(* IEC 61131-3 sources: A_BST22/, 17 files *)

(* ---- PLC_Arcade_System_ST.st ---- *)
// Sysmac Studio Structured Text - PLC Arcade System
// Omron NX102 PLC Implementation

// Global Variables Declaration
VAR_GLOBAL
    // ============================================================================
    // INPUT MAPPING (Contacts)
    // ============================================================================
    IBTN_R AT %IX0.0: BOOL;      // Red button - DI0
    IBTN_B AT %IX0.2: BOOL;      // Blue button - DI2
    IBTN_Y AT %IX0.4: BOOL;      // Yellow button - DI4
    ISEL_LT AT %IX0.3: BOOL;     // Simon Says selector - DI3 (Yellow wire)
    ISEL_R AT %IX0.5: BOOL;      // Reaction Game selector - DI5 (Green wire)
    IBTN_M AT %IX0.1: BOOL;      // Main button - DI1 (Brown wire)

    // ============================================================================
    // OUTPUT MAPPING (LEDs)
    // ============================================================================
    OLED_R AT %QX0.1: BOOL;      // Red LED - DO1
    OLED_B AT %QX0.3: BOOL;      // Blue LED - DO3
    OLED_Y AT %QX0.5: BOOL;      // Yellow LED - DO5
    OLED_MAIN AT %QX0.0: BOOL;   // Main LED - DO0 (White wire)

    // ============================================================================
    // SYSTEM CONTROL VARIABLES
    // ============================================================================
    SystemActive: BOOL := FALSE;
    GameRunning: BOOL := FALSE;
    ModeLocked: BOOL := FALSE;
    EmergencyStop: BOOL := FALSE;

    // Mode Selection
    CurrentMode: INT := 0;  // 0=Simon Says, 1=Reaction Game, 2=Idle
    PreviousMode: INT := 0;

    // Button States (Debounced)
    BtnR_State: BOOL := FALSE;
    BtnB_State: BOOL := FALSE;
    BtnY_State: BOOL := FALSE;
    BtnM_State: BOOL := FALSE;

    // Button Edge Detection
    BtnR_Rising: BOOL := FALSE;
    BtnB_Rising: BOOL := FALSE;
    BtnY_Rising: BOOL := FALSE;
    BtnM_Rising: BOOL := FALSE;

    // Previous Button States for Edge Detection
    PrevBtnR: BOOL := FALSE;
    PrevBtnB: BOOL := FALSE;
    PrevBtnY: BOOL := FALSE;
    PrevBtnM: BOOL := FALSE;

    // ============================================================================
    // DEBOUNCE TIMERS (Sysmac Studio TON)
    // ============================================================================
    DebounceTimer: TON;
    ModeLockTimer: TON;

    // ============================================================================
    // CONTINUOUS RANDOM GENERATOR VARIABLES
    // ============================================================================
    RandomGenActive: BOOL := FALSE;
    RandomGenRunning: BOOL := FALSE;
    RandomCounter: INT := 0;
    OutputSelect: INT := 0;

    // Random Generator Outputs
    RandomOut1: BOOL := FALSE;
    RandomOut2: BOOL := FALSE;
    RandomOut3: BOOL := FALSE;

    // ============================================================================
    // SIMON SAYS GAME VARIABLES
    // ============================================================================
    SimonActive: BOOL := FALSE;
    SimonGameOver: BOOL := FALSE;
    SimonState: INT := 0;  // 0=Off, 1=Init, 2=Generate, 3=Show, 4=Input, 5=Check, 6=Complete

    SimonSequence: ARRAY[1..20] OF INT := [0,0,0,0,0,0,0,0,0,0,0,0,0,0,0,0,0,0,0,0];
    SequenceLength: INT := 1;
    CurrentStep: INT := 0;
    PlayerInputStep: INT := 0;

    SimonScore: INT := 0;
    SimonLevel: INT := 1;

    // Simon Says Timers
    SimonSequenceTimer: TON;
    SimonInputTimer: TON;
    SimonPauseTimer: TON;

    // Simon Says Outputs
    SimonOut1: BOOL := FALSE;
    SimonOut2: BOOL := FALSE;
    SimonOut3: BOOL := FALSE;

    // ============================================================================
    // REACTION GAME VARIABLES
    // ============================================================================
    ReactionActive: BOOL := FALSE;
    ReactionGameOver: BOOL := FALSE;
    ReactionState: INT := 0;  // 0=Off, 1=Wait, 2=Show, 3=Score

    ReactionStartTime: INT := 0;
    ReactionEndTime: INT := 0;
    ReactionScore: INT := 0;
    ReactionTarget: INT := 0;  // Which LED to light up (1,2,3)

    // Reaction Game Timers
    ReactionWaitTimer: TON;
    ReactionShowTimer: TON;

    // Reaction Game Outputs
    ReactionOut1: BOOL := FALSE;
    ReactionOut2: BOOL := FALSE;
    ReactionOut3: BOOL := FALSE;

    // ============================================================================
    // OUTPUT MAPPER VARIABLES
    // ============================================================================
    OutputPriority: INT := 0;  // 0=Off, 1=Game, 2=Status, 3=Emergency
    OutputConflict: BOOL := FALSE;
    SafetyInterlock: BOOL := TRUE;
    SystemHealthy: BOOL := TRUE;

    // Status Outputs
    StatusOut1: BOOL := FALSE;
    StatusOut2: BOOL := FALSE;
    StatusOut3: BOOL := FALSE;

    // Emergency Outputs
    EmergencyOut1: BOOL := FALSE;
    EmergencyOut2: BOOL := FALSE;
    EmergencyOut3: BOOL := FALSE;

    // ============================================================================
    // TIMING VARIABLES (Sysmac Studio TON)
    // ============================================================================
    SystemTimer: TON;
    BlinkTimer: TON;

    // ============================================================================
    // DIAGNOSTIC VARIABLES
    // ============================================================================
    ConflictCounter: INT := 0;
    SafetyFailureCounter: INT := 0;
    SystemFailureCounter: INT := 0;

END_VAR

// ============================================================================
// MAIN PROGRAM LOGIC
// ============================================================================

// Note: Input mapping is done directly in VAR_GLOBAL with AT %IX addresses
// No additional mapping needed - inputs are automatically read from hardware

// Button Edge Detection
BtnR_Rising := IBTN_R AND NOT PrevBtnR;
BtnB_Rising := IBTN_B AND NOT PrevBtnB;
BtnY_Rising := IBTN_Y AND NOT PrevBtnY;
BtnM_Rising := IBTN_M AND NOT PrevBtnM;

PrevBtnR := IBTN_R;
PrevBtnB := IBTN_B;
PrevBtnY := IBTN_Y;
PrevBtnM := IBTN_M;

// Button Debouncing (Sysmac Studio TON syntax)
DebounceTimer(IN := IBTN_R OR IBTN_B OR IBTN_Y OR IBTN_M, PT := T#50MS);

IF DebounceTimer.Q THEN
    BtnR_State := IBTN_R;
    BtnB_State := IBTN_B;
    BtnY_State := IBTN_Y;
    BtnM_State := IBTN_M;
    DebounceTimer(IN := FALSE, PT := T#0MS);  // Reset timer
END_IF;

// Mode Selection Logic
PreviousMode := CurrentMode;

IF ISEL_LT THEN
    CurrentMode := 0;  // Simon Says
ELSIF ISEL_R THEN
    CurrentMode := 1;  // Reaction Game
ELSE
    CurrentMode := 2;  // Idle Mode
END_IF;

// Mode Lock Logic
IF BtnM_Rising AND NOT ModeLocked THEN
    ModeLocked := TRUE;
    ModeLockTimer(IN := FALSE, PT := T#0MS);
ELSIF BtnM_Rising AND ModeLocked THEN
    ModeLocked := FALSE;
END_IF;

// System Activation
IF ModeLocked AND BtnM_Rising THEN
    GameRunning := TRUE;
    SystemActive := TRUE;
END_IF;

// Emergency Stop
IF EmergencyStop THEN
    GameRunning := FALSE;
    SystemActive := FALSE;
    ModeLocked := FALSE;
    OutputPriority := 3;  // Emergency priority
END_IF;

// ============================================================================
// CONTINUOUS RANDOM GENERATOR
// ============================================================================

RandomGenActive := SystemActive;

// Random Generator Timer (Sysmac Studio TON syntax)
SystemTimer(IN := RandomGenActive, PT := T#100MS);

// Increment Counter
IF SystemTimer.Q THEN
    SystemTimer(IN := FALSE, PT := T#0MS);  // Reset timer
    RandomCounter := RandomCounter + 1;
    IF RandomCounter >= 1000 THEN
        RandomCounter := 0;
    END_IF;
END_IF;

// Calculate Output Selection
OutputSelect := RandomCounter MOD 3;
RandomGenRunning := RandomGenActive;

// Set Random Outputs
RandomOut1 := RandomGenRunning AND (OutputSelect = 0);
RandomOut2 := RandomGenRunning AND (OutputSelect = 1);
RandomOut3 := RandomGenRunning AND (OutputSelect = 2);

// ============================================================================
// SIMON SAYS GAME LOGIC
// ============================================================================

SimonActive := (CurrentMode = 0) AND GameRunning;

// Simon Says State Machine
CASE SimonState OF
    0:  // Game Off
        IF SimonActive THEN
            SimonState := 1;
            SimonScore := 0;
            SimonLevel := 1;
            SequenceLength := 1;
            SimonGameOver := FALSE;
        END_IF;

    1:  // Initialize Game
        CurrentStep := 0;
        PlayerInputStep := 0;
        SimonSequenceTimer(IN := FALSE, PT := T#0MS);
        SimonInputTimer(IN := FALSE, PT := T#0MS);
        SimonPauseTimer(IN := FALSE, PT := T#0MS);
        SimonState := 2;

    2:  // Generate Sequence
        FOR i := 1 TO SequenceLength DO
            SimonSequence[i] := (RandomCounter + i) MOD 3 + 1;
        END_FOR;
        SimonState := 3;

    3:  // Show Sequence
        IF CurrentStep < SequenceLength THEN
            SimonSequenceTimer(IN := TRUE, PT := T#500MS);
            IF SimonSequenceTimer.Q THEN
                SimonSequenceTimer(IN := FALSE, PT := T#0MS);  // Reset timer
                CurrentStep := CurrentStep + 1;
            END_IF;
        ELSE
            SimonPauseTimer(IN := TRUE, PT := T#1000MS);
            IF SimonPauseTimer.Q THEN
                SimonPauseTimer(IN := FALSE, PT := T#0MS);  // Reset timer
                CurrentStep := 0;
                PlayerInputStep := 0;
                SimonState := 4;
            END_IF;
        END_IF;

    4:  // Wait for Player Input
        SimonInputTimer(IN := TRUE, PT := T#5000MS);

        // Check for player input
        IF BtnR_Rising THEN
            IF SimonSequence[PlayerInputStep + 1] = 1 THEN
                PlayerInputStep := PlayerInputStep + 1;
            ELSE
                SimonGameOver := TRUE;
                SimonState := 6;
            END_IF;
        ELSIF BtnB_Rising THEN
            IF SimonSequence[PlayerInputStep + 1] = 2 THEN
                PlayerInputStep := PlayerInputStep + 1;
            ELSE
                SimonGameOver := TRUE;
                SimonState := 6;
            END_IF;
        ELSIF BtnY_Rising THEN
            IF SimonSequence[PlayerInputStep + 1] = 3 THEN
                PlayerInputStep := PlayerInputStep + 1;
            ELSE
                SimonGameOver := TRUE;
                SimonState := 6;
            END_IF;
        END_IF;

        // Check if input complete or timeout
        IF PlayerInputStep >= SequenceLength THEN
            SimonScore := SimonScore + (SequenceLength * 10);
            SequenceLength := SequenceLength + 1;
            SimonState := 2;  // Generate next sequence
        ELSIF SimonInputTimer.Q THEN
            SimonGameOver := TRUE;
            SimonState := 6;
        END_IF;

    5:  // Check Input (Not used in this implementation)
        SimonState := 6;

    6:  // Game Complete
        SimonInputTimer(IN := FALSE, PT := T#0MS);  // Reset timer
        IF NOT SimonActive THEN
            SimonState := 0;
        END_IF;
END_CASE;

// Simon Says Output Control
SimonOut1 := (SimonState = 3) AND (CurrentStep <= SequenceLength) AND (SimonSequence[CurrentStep] = 1);
SimonOut2 := (SimonState = 3) AND (CurrentStep <= SequenceLength) AND (SimonSequence[CurrentStep] = 2);
SimonOut3 := (SimonState = 3) AND (CurrentStep <= SequenceLength) AND (SimonSequence[CurrentStep] = 3);

// Add player input feedback
SimonOut1 := SimonOut1 OR ((SimonState = 4) AND BtnR_State);
SimonOut2 := SimonOut2 OR ((SimonState = 4) AND BtnB_State);
SimonOut3 := SimonOut3 OR ((SimonState = 4) AND BtnY_State);

// ============================================================================
// REACTION GAME LOGIC
// ============================================================================

ReactionActive := (CurrentMode = 1) AND GameRunning;

// Reaction Game State Machine
CASE ReactionState OF
    0:  // Game Off
        IF ReactionActive THEN
            ReactionState := 1;
            ReactionScore := 0;
            ReactionGameOver := FALSE;
        END_IF;

    1:  // Wait Phase
        ReactionWaitTimer(IN := TRUE, PT := T#2000MS + (RandomCounter MOD 3000MS));
        IF ReactionWaitTimer.Q THEN
            ReactionWaitTimer(IN := FALSE, PT := T#0MS);  // Reset timer
            ReactionTarget := (RandomCounter MOD 3) + 1;
            ReactionState := 2;
        END_IF;

    2:  // Show Target
        ReactionShowTimer(IN := TRUE, PT := T#1000MS);

        // Check for player reaction
        IF (ReactionTarget = 1) AND BtnR_Rising THEN
            ReactionEndTime := 1000 - ReactionShowTimer.ET;
            ReactionScore := ReactionEndTime;
            ReactionState := 3;
        ELSIF (ReactionTarget = 2) AND BtnB_Rising THEN
            ReactionEndTime := 1000 - ReactionShowTimer.ET;
            ReactionScore := ReactionEndTime;
            ReactionState := 3;
        ELSIF (ReactionTarget = 3) AND BtnY_Rising THEN
            ReactionEndTime := 1000 - ReactionShowTimer.ET;
            ReactionScore := ReactionEndTime;
            ReactionState := 3;
        ELSIF ReactionShowTimer.Q THEN
            ReactionGameOver := TRUE;
            ReactionState := 3;
        END_IF;

    3:  // Score Phase
        IF NOT ReactionActive THEN
            ReactionState := 0;
        ELSIF BtnM_Rising THEN
            ReactionState := 1;  // Start new round
        END_IF;
END_CASE;

// Reaction Game Output Control
ReactionOut1 := (ReactionState = 2) AND (ReactionTarget = 1);
ReactionOut2 := (ReactionState = 2) AND (ReactionTarget = 2);
ReactionOut3 := (ReactionState = 2) AND (ReactionTarget = 3);

// ============================================================================
// OUTPUT MAPPER AND SAFETY LOGIC
// ============================================================================

// Detect Output Conflicts
OutputConflict := (SimonActive AND ReactionActive) OR
                  (SimonActive AND (CurrentMode = 2)) OR
                  (ReactionActive AND (CurrentMode = 2));

// Output Priority Control
IF EmergencyStop THEN
    OutputPriority := 3;  // Emergency
ELSIF NOT SystemHealthy THEN
    OutputPriority := 3;  // Emergency
ELSIF OutputConflict THEN
    OutputPriority := 3;  // Emergency
ELSIF GameRunning THEN
    OutputPriority := 1;  // Game
ELSIF SystemActive THEN
    OutputPriority := 2;  // Status
ELSE
    OutputPriority := 0;  // Off
END_IF;

// Status Outputs
StatusOut1 := SystemActive;
StatusOut2 := GameRunning;
StatusOut3 := OutputConflict OR NOT SystemHealthy;

// Emergency Outputs
EmergencyOut1 := EmergencyStop;
EmergencyOut2 := NOT SystemHealthy;
EmergencyOut3 := OutputConflict;

// Final Output Mapping
CASE OutputPriority OF
    0:  // System Off
        OLED_R := FALSE;
        OLED_B := FALSE;
        OLED_Y := FALSE;
        OLED_MAIN := FALSE;

    1:  // Game Outputs
        IF CurrentMode = 0 THEN  // Simon Says
            OLED_R := SimonOut1;
            OLED_B := SimonOut2;
            OLED_Y := SimonOut3;
        ELSIF CurrentMode = 1 THEN  // Reaction Game
            OLED_R := ReactionOut1;
            OLED_B := ReactionOut2;
            OLED_Y := ReactionOut3;
        ELSE  // Idle Mode
            OLED_R := RandomOut1;
            OLED_B := RandomOut2;
            OLED_Y := RandomOut3;
        END_IF;
        OLED_MAIN := GameRunning;

    2:  // Status Outputs
        OLED_R := StatusOut1;
        OLED_B := StatusOut2;
        OLED_Y := StatusOut3;
        OLED_MAIN := ModeLocked;

    3:  // Emergency Outputs
        OLED_R := EmergencyOut1;
        OLED_B := EmergencyOut2;
        OLED_Y := EmergencyOut3;
        OLED_MAIN := FALSE;
END_CASE;

// Note: Output mapping is done directly in VAR_GLOBAL with AT %QX addresses
// No additional mapping needed - outputs are automatically written to hardware
// OLED_R AT %QX0.1, OLED_B AT %QX0.3, OLED_Y AT %QX0.5, OLED_MAIN AT %QX0.0

// ============================================================================
// DIAGNOSTIC AND MONITORING
// ============================================================================

// Count Conflicts
IF OutputConflict THEN
    ConflictCounter := ConflictCounter + 1;
END_IF;

// Count Safety Failures
IF NOT SystemHealthy THEN
    SafetyFailureCounter := SafetyFailureCounter + 1;
END_IF;

// System Health Check
SystemHealthy := TRUE;  // Placeholder - implement actual health checks

// ============================================================================
// END OF PROGRAM
// ============================================================================

(* ---- HandleButtonPress.st ---- *)
FUNCTION HandleButtonPress : BOOL
VAR_INPUT
    ButtonPressed : BOOL;           // TRUE if this button was pressed
    ExpectedLED : INT;             // The LED number that should be lit (1=Yellow, 2=Blue, 3=Red)
    CurrentLED : INT;              // The currently lit LED number
END_VAR

VAR_IN_OUT
    Score : INT;                   // Player's current score
    GameActive : BOOL;             // Game state flag
    GameOver_Active : BOOL;        // Game over state flag
    LEDActive : BOOL;              // LED phase active flag
    GapActive : BOOL;              // Gap phase active flag
    HighScore : INT;               // High score tracking
    GameOver_Step : INT;           // Game over sequence step
    T_LED_On : TON;                // LED timer
    T_Gap : TON;                   // Gap timer
    T_Seq : TON;                   // Sequence timer
    Rand_Gen : FB_Random;          // Random number generator
    RandN : REAL;                  // Random number output
END_VAR

// Function returns TRUE if button was handled (pressed)
HandleButtonPress := ButtonPressed;

IF ButtonPressed THEN
    IF CurrentLED = ExpectedLED THEN
        // Correct button pressed - add point and continue
        Score := Score + 1;
        LEDActive := FALSE;
        GapActive := TRUE;
        T_LED_On(IN := FALSE);

        // Generate next random gap duration
        Rand_Gen(Execute := TRUE, Seed := 0, Rnd => RandN);
        T_Gap(IN := FALSE);
        IF RandN < 0.2 THEN
            T_Gap(PT := t#500ms);
        ELSIF RandN < 0.4 THEN
            T_Gap(PT := t#750ms);
        ELSIF RandN < 0.6 THEN
            T_Gap(PT := t#1000ms);
        ELSIF RandN < 0.8 THEN
            T_Gap(PT := t#1250ms);
        ELSE
            T_Gap(PT := t#1500ms);
        END_IF;
    ELSE
        // Wrong button pressed - game over
        GameActive := FALSE;
        GameOver_Active := TRUE;
        GameOver_Step := 0;
        T_Seq(IN := FALSE, PT := t#300ms);
        LEDActive := FALSE;
        GapActive := FALSE;
        T_LED_On(IN := FALSE);
        T_Gap(IN := FALSE);

        // Update high score if needed
        IF Score > HighScore THEN
            HighScore := Score;
        END_IF;
    END_IF;
END_IF;

END_FUNCTION

(* ---- FB_CheckButtonPress.st ---- *)
FUNCTION_BLOCK FB_CheckButtonPress
VAR_INPUT
    ButtonPressed : BOOL;          // Trigger for this button
    ExpectedLED : INT;             // Which LED should be lit (1=Yellow, 2=Blue, 3=Red)
    CurrentLED : INT;              // Which LED is actually lit
    Score : INT;                   // Current score
    HighScore : INT;               // Current high score
END_VAR

VAR_OUTPUT
    IsCorrect : BOOL;              // TRUE if correct button pressed
    IsWrong : BOOL;                // TRUE if wrong button pressed
    NewScore : INT;                // Updated score
    NewHighScore : INT;            // Updated high score
    NextGapTime : TIME;            // Random gap time for next round
    EndGame : BOOL;                // Signal to end the game
    ContinueGame : BOOL;           // Signal to continue to next round
END_VAR

VAR
    Rand_Gen : FB_RandomGenerator; // Random number generator (adjust to your actual FB name)
    RandN : REAL;
END_VAR

// Initialize outputs
IsCorrect := FALSE;
IsWrong := FALSE;
NewScore := Score;
NewHighScore := HighScore;
EndGame := FALSE;
ContinueGame := FALSE;

// Check if button was pressed
IF ButtonPressed THEN
    // Check if it's the correct button
    IF CurrentLED = ExpectedLED THEN
        // Correct button pressed
        IsCorrect := TRUE;
        ContinueGame := TRUE;
        NewScore := Score + 1;

        // Generate next random gap time
        Rand_Gen(Execute := TRUE, Seed := 0, Rnd => RandN);
        IF RandN < 0.2 THEN
            NextGapTime := t#500ms;
        ELSIF RandN < 0.4 THEN
            NextGapTime := t#750ms;
        ELSIF RandN < 0.6 THEN
            NextGapTime := t#1000ms;
        ELSIF RandN < 0.8 THEN
            NextGapTime := t#1250ms;
        ELSE
            NextGapTime := t#1500ms;
        END_IF;
    ELSE
        // Wrong button pressed - game over
        IsWrong := TRUE;
        EndGame := TRUE;

        // Update high score if needed
        IF Score > HighScore THEN
            NewHighScore := Score;
        ELSE
            NewHighScore := HighScore;
        END_IF;
    END_IF;
END_IF;

END_FUNCTION_BLOCK

(* ---- FB_RandomGenerator.st ---- *)
(* ====================================================================
   FUNCTION BLOCK: Random Number Generator for Simon Says
   Generates pseudo-random numbers 1-3 for button selection
   ==================================================================== *)

FUNCTION_BLOCK FB_RandomGenerator
VAR_INPUT
    Generate : BOOL;        (* Trigger to generate new random number *)
    Reset : BOOL;           (* Reset seed to initial value *)
    MaxValue : INT := 3;    (* Maximum value (3 for 3 buttons, 4 for 4 buttons) *)
END_VAR

VAR_OUTPUT
    RandomValue : INT;      (* Output: 1 to MaxValue *)
    Done : BOOL;           (* Pulse when new number generated *)
END_VAR

VAR
    Seed : DINT := 12345;  (* Internal seed value *)
    LastGenerate : BOOL;   (* Edge detection *)
    PulseTimer : TON;      (* Timer for done pulse *)
END_VAR

(* Reset seed if requested *)
IF Reset THEN
    Seed := 12345;
    RandomValue := 0;
    Done := FALSE;
END_IF;

(* Detect rising edge of Generate signal *)
IF Generate AND NOT LastGenerate THEN
    (* Linear Congruential Generator algorithm *)
    Seed := (Seed * 1103515245 + 12345) MOD 2147483648;

    (* Convert to desired range (1 to MaxValue) *)
    RandomValue := (ABS(Seed) MOD MaxValue) + 1;

    (* Trigger done pulse *)
    Done := TRUE;
    PulseTimer(IN := TRUE, PT := T#100MS);
END_IF;

(* Clear done pulse after timer *)
PulseTimer(IN := PulseTimer.IN, PT := T#100MS);
IF PulseTimer.Q THEN
    Done := FALSE;
    PulseTimer(IN := FALSE);
END_IF;

(* Update edge detection *)
LastGenerate := Generate;

END_FUNCTION_BLOCK

(* ---- FB_SimonSays.st ---- *)
(* ====================================================================== *)
(* Function Block: FB_SimonSays                                          *)
(* Simon Says Game Logic for Omron NX102                                *)
(* ====================================================================== *)

FUNCTION_BLOCK FB_SimonSays

VAR_INPUT
    (* Button Inputs *)
    i_YellowButton : BOOL;     (* Yellow button contact *)
    i_BlueButton : BOOL;       (* Blue button contact *)
    i_RedButton : BOOL;         (* Red button contact *)
    i_StartButton : BOOL;       (* Start/Stop button *)
    i_Reset : BOOL;             (* Reset game *)

    (* Game Parameters *)
    i_MaxLevel : INT := 10;    (* Maximum sequence length *)
    i_ShowTime : TIME := T#500MS;   (* LED display time *)
    i_GapTime : TIME := T#200MS;    (* Gap between LEDs *)
    i_InputTimeout : TIME := T#3S;  (* Player input timeout *)
END_VAR

VAR_OUTPUT
    (* LED Outputs *)
    q_YellowLED : BOOL;        (* Yellow button LED *)
    q_BlueLED : BOOL;          (* Blue button LED *)
    q_RedLED : BOOL;           (* Red button LED *)

    (* Status Outputs *)
    q_GameActive : BOOL;        (* Game is active *)
    q_CurrentLevel : INT;       (* Current level *)
    q_GameWon : BOOL;          (* Player won *)
    q_GameLost : BOOL;         (* Player lost *)
    q_State : INT;             (* Current state for diagnostics *)
END_VAR

VAR
    (* Internal State Machine *)
    State : INT := 0;
    NextState : INT := 0;

    (* Sequence Storage *)
    Sequence : ARRAY[0..49] OF INT;
    Level : INT := 0;
    SeqIndex : INT := 0;
    InputIndex : INT := 0;

    (* Timers *)
    tmr_Show : TON;
    tmr_Gap : TON;
    tmr_Input : TON;
    tmr_GameOver : TON;
    tmr_Blink : TON;

    (* Edge Detection *)
    rtrig_Yellow : R_TRIG;
    rtrig_Blue : R_TRIG;
    rtrig_Red : R_TRIG;
    rtrig_Start : R_TRIG;

    (* Flags *)
    ShowingLED : BOOL := FALSE;
    InGap : BOOL := FALSE;
    InputReceived : BOOL := FALSE;
    CorrectInput : BOOL := FALSE;

    (* Random Generation *)
    RandomSeed : DINT := 0;
    RandomValue : INT := 0;

    (* Temporary Variables *)
    i : INT;
    BlinkState : BOOL := FALSE;
END_VAR

(* ====================================================================== *)
(* MAIN LOGIC                                                            *)
(* ====================================================================== *)

(* Edge Detection *)
rtrig_Yellow(CLK := i_YellowButton);
rtrig_Blue(CLK := i_BlueButton);
rtrig_Red(CLK := i_RedButton);
rtrig_Start(CLK := i_StartButton);

(* Update Random Seed *)
RandomSeed := RandomSeed + 1;
IF RandomSeed > 100000 THEN
    RandomSeed := 1;
END_IF;

(* Reset Logic *)
IF i_Reset THEN
    State := 0;
    Level := 0;
    SeqIndex := 0;
    InputIndex := 0;
    q_YellowLED := FALSE;
    q_BlueLED := FALSE;
    q_RedLED := FALSE;
    q_GameActive := FALSE;
    q_GameWon := FALSE;
    q_GameLost := FALSE;
    ShowingLED := FALSE;
    InGap := FALSE;
    RETURN;
END_IF;

(* State Machine *)
CASE State OF

    (* ====================================================================== *)
    0: (* IDLE STATE *)
    (* ====================================================================== *)
        q_GameActive := FALSE;
        q_YellowLED := FALSE;
        q_BlueLED := FALSE;
        q_RedLED := FALSE;
        q_GameWon := FALSE;
        q_GameLost := FALSE;

        IF rtrig_Start.Q THEN
            (* Initialize new game *)
            Level := 1;
            SeqIndex := 0;
            InputIndex := 0;

            (* Generate first random button *)
            RandomValue := INT(RandomSeed MOD 3) + 1;
            Sequence[0] := RandomValue;

            (* Start game *)
            q_GameActive := TRUE;
            State := 1;
        END_IF;

    (* ====================================================================== *)
    1: (* SHOW SEQUENCE STATE *)
    (* ====================================================================== *)
        IF SeqIndex < Level THEN
            IF NOT ShowingLED AND NOT InGap THEN
                (* Start showing next LED *)
                ShowingLED := TRUE;
                tmr_Show(IN := FALSE);
                tmr_Show(IN := TRUE, PT := i_ShowTime);

                (* Turn on appropriate LED *)
                CASE Sequence[SeqIndex] OF
                    1: q_YellowLED := TRUE;
                    2: q_BlueLED := TRUE;
                    3: q_RedLED := TRUE;
                END_CASE;
            END_IF;

            (* Handle LED display timing *)
            IF ShowingLED THEN
                tmr_Show(IN := TRUE, PT := i_ShowTime);
                IF tmr_Show.Q THEN
                    (* Turn off LEDs *)
                    q_YellowLED := FALSE;
                    q_BlueLED := FALSE;
                    q_RedLED := FALSE;
                    ShowingLED := FALSE;
                    InGap := TRUE;
                    tmr_Gap(IN := FALSE);
                    tmr_Gap(IN := TRUE, PT := i_GapTime);
                END_IF;
            END_IF;

            (* Handle gap timing *)
            IF InGap THEN
                tmr_Gap(IN := TRUE, PT := i_GapTime);
                IF tmr_Gap.Q THEN
                    InGap := FALSE;
                    SeqIndex := SeqIndex + 1;
                END_IF;
            END_IF;
        ELSE
            (* Sequence display complete *)
            SeqIndex := 0;
            InputIndex := 0;
            State := 2;
            tmr_Input(IN := FALSE);
            tmr_Input(IN := TRUE, PT := i_InputTimeout);
        END_IF;

    (* ====================================================================== *)
    2: (* WAIT FOR PLAYER INPUT STATE *)
    (* ====================================================================== *)
        (* Check for timeout *)
        tmr_Input(IN := TRUE, PT := i_InputTimeout);
        IF tmr_Input.Q THEN
            (* Timeout - player loses *)
            State := 4;
            tmr_GameOver(IN := FALSE);
            tmr_GameOver(IN := TRUE, PT := T#2S);
        END_IF;

        (* Process button inputs *)
        InputReceived := FALSE;
        CorrectInput := FALSE;

        IF rtrig_Yellow.Q THEN
            InputReceived := TRUE;
            q_YellowLED := TRUE;
            IF Sequence[InputIndex] = 1 THEN
                CorrectInput := TRUE;
            END_IF;
        ELSIF rtrig_Blue.Q THEN
            InputReceived := TRUE;
            q_BlueLED := TRUE;
            IF Sequence[InputIndex] = 2 THEN
                CorrectInput := TRUE;
            END_IF;
        ELSIF rtrig_Red.Q THEN
            InputReceived := TRUE;
            q_RedLED := TRUE;
            IF Sequence[InputIndex] = 3 THEN
                CorrectInput := TRUE;
            END_IF;
        END_IF;

        (* Turn off LEDs when buttons released *)
        IF NOT i_YellowButton THEN q_YellowLED := FALSE; END_IF;
        IF NOT i_BlueButton THEN q_BlueLED := FALSE; END_IF;
        IF NOT i_RedButton THEN q_RedLED := FALSE; END_IF;

        (* Process input result *)
        IF InputReceived THEN
            IF CorrectInput THEN
                (* Correct input *)
                InputIndex := InputIndex + 1;
                tmr_Input(IN := FALSE);
                tmr_Input(IN := TRUE, PT := i_InputTimeout);

                (* Check if sequence complete *)
                IF InputIndex >= Level THEN
                    IF Level >= i_MaxLevel THEN
                        (* Player wins! *)
                        State := 3;
                        tmr_GameOver(IN := FALSE);
                        tmr_GameOver(IN := TRUE, PT := T#3S);
                    ELSE
                        (* Next level *)
                        Level := Level + 1;
                        RandomValue := INT((RandomSeed * Level) MOD 3) + 1;
                        Sequence[Level - 1] := RandomValue;

                        (* Small delay before showing new sequence *)
                        tmr_Gap(IN := FALSE);
                        InGap := TRUE;
                        tmr_Gap(IN := TRUE, PT := T#1S);

                        IF tmr_Gap.Q THEN
                            InGap := FALSE;
                            SeqIndex := 0;
                            State := 1;
                        END_IF;
                    END_IF;
                END_IF;
            ELSE
                (* Wrong input - player loses *)
                State := 4;
                tmr_GameOver(IN := FALSE);
                tmr_GameOver(IN := TRUE, PT := T#2S);
            END_IF;
        END_IF;

    (* ====================================================================== *)
    3: (* GAME WON STATE *)
    (* ====================================================================== *)
        q_GameWon := TRUE;

        (* Victory light show *)
        tmr_Blink(IN := TRUE, PT := T#200MS);
        IF tmr_Blink.Q THEN
            tmr_Blink(IN := FALSE);
            BlinkState := NOT BlinkState;
        END_IF;

        IF BlinkState THEN
            q_YellowLED := TRUE;
            q_BlueLED := TRUE;
            q_RedLED := TRUE;
        ELSE
            q_YellowLED := FALSE;
            q_BlueLED := FALSE;
            q_RedLED := FALSE;
        END_IF;

        (* Check if celebration complete *)
        tmr_GameOver(IN := TRUE, PT := T#3S);
        IF tmr_GameOver.Q THEN
            State := 0;
        END_IF;

    (* ====================================================================== *)
    4: (* GAME LOST STATE *)
    (* ====================================================================== *)
        q_GameLost := TRUE;

        (* Flash red LED *)
        tmr_Blink(IN := TRUE, PT := T#300MS);
        IF tmr_Blink.Q THEN
            tmr_Blink(IN := FALSE);
            BlinkState := NOT BlinkState;
        END_IF;

        q_RedLED := BlinkState;
        q_YellowLED := FALSE;
        q_BlueLED := FALSE;

        (* Check if game over display complete *)
        tmr_GameOver(IN := TRUE, PT := T#2S);
        IF tmr_GameOver.Q THEN
            State := 0;
        END_IF;

END_CASE;

(* Update outputs *)
q_State := State;
q_CurrentLevel := Level;

END_FUNCTION_BLOCK

(* ---- reaction_game_optimized.st ---- *)
// OPTIMIZED REACTION GAME LOGIC WITH UNIFIED BUTTON HANDLING

// =============================================================================
// UNIFIED BUTTON HANDLER FUNCTION BLOCK
// =============================================================================

FUNCTION_BLOCK FB_ProcessButtonInput
VAR_INPUT
    // Button triggers
    Yellow_Pressed : BOOL;
    Blue_Pressed : BOOL;
    Red_Pressed : BOOL;

    // Game state
    CurrentLED : INT;          // Which LED is on (1=Y, 2=B, 3=R, 0=none)
    IsGapPhase : BOOL;         // TRUE if in gap phase
    IsLEDPhase : BOOL;         // TRUE if in LED phase
END_VAR

VAR_OUTPUT
    ButtonPressed : INT;       // Which button was pressed (1=Y, 2=B, 3=R, 0=none)
    IsCorrect : BOOL;         // TRUE if correct button
    IsError : BOOL;           // TRUE if wrong button or wrong timing
    ShouldAddPoint : BOOL;    // TRUE to increment score
END_VAR

// Reset outputs
ButtonPressed := 0;
IsCorrect := FALSE;
IsError := FALSE;
ShouldAddPoint := FALSE;

// Determine which button was pressed
IF Yellow_Pressed THEN
    ButtonPressed := 1;
ELSIF Blue_Pressed THEN
    ButtonPressed := 2;
ELSIF Red_Pressed THEN
    ButtonPressed := 3;
END_IF;

// Process button press
IF ButtonPressed > 0 THEN
    IF IsGapPhase THEN
        // Any button during gap = error
        IsError := TRUE;
    ELSIF IsLEDPhase THEN
        IF ButtonPressed = CurrentLED THEN
            // Correct!
            IsCorrect := TRUE;
            ShouldAddPoint := TRUE;
        ELSE
            // Wrong button
            IsError := TRUE;
        END_IF;
    END_IF;
END_IF;

END_FUNCTION_BLOCK

// =============================================================================
// HELPER FUNCTION FOR RANDOM GAP GENERATION
// =============================================================================

FUNCTION F_GetRandomGapTime : TIME
VAR_INPUT
    RandomValue : REAL;
END_VAR

IF RandomValue < 0.2 THEN
    F_GetRandomGapTime := t#500ms;
ELSIF RandomValue < 0.4 THEN
    F_GetRandomGapTime := t#750ms;
ELSIF RandomValue < 0.6 THEN
    F_GetRandomGapTime := t#1000ms;
ELSIF RandomValue < 0.8 THEN
    F_GetRandomGapTime := t#1250ms;
ELSE
    F_GetRandomGapTime := t#1500ms;
END_IF;

END_FUNCTION

// =============================================================================
// HELPER FUNCTION BLOCK FOR TRANSITIONING TO GAME OVER
// =============================================================================

FUNCTION_BLOCK FB_TriggerGameOver
VAR_INPUT
    Execute : BOOL;
    CurrentScore : INT;
END_VAR

VAR_IN_OUT
    GameActive : BOOL;
    GameOver_Active : BOOL;
    GameOver_Step : INT;
    LEDActive : BOOL;
    GapActive : BOOL;
    HighScore : INT;
END_VAR

VAR_OUTPUT
    Done : BOOL;
END_VAR

Done := FALSE;

IF Execute THEN
    // Update game state
    GameActive := FALSE;
    GameOver_Active := TRUE;
    GameOver_Step := 0;
    LEDActive := FALSE;
    GapActive := FALSE;

    // Check high score
    IF CurrentScore > HighScore THEN
        HighScore := CurrentScore;
    END_IF;

    Done := TRUE;
END_IF;

END_FUNCTION_BLOCK

// =============================================================================
// HELPER FUNCTION BLOCK FOR STARTING NEXT ROUND
// =============================================================================

FUNCTION_BLOCK FB_PrepareNextRound
VAR_INPUT
    Execute : BOOL;
END_VAR

VAR_IN_OUT
    Score : INT;
    LEDActive : BOOL;
    GapActive : BOOL;
END_VAR

VAR_OUTPUT
    NewGapTime : TIME;
    Done : BOOL;
END_VAR

VAR
    LocalRand : REAL;
END_VAR

Done := FALSE;

IF Execute THEN
    // Update score
    Score := Score + 1;

    // Switch to gap phase
    LEDActive := FALSE;
    GapActive := TRUE;

    // Generate random gap time
    Rand_Gen(Execute := TRUE, Seed := 0, Rnd => LocalRand);
    NewGapTime := F_GetRandomGapTime(RandomValue := LocalRand);

    Done := TRUE;
END_IF;

END_FUNCTION_BLOCK

// =============================================================================
// MAIN PROGRAM - OPTIMIZED VERSION
// =============================================================================

PROGRAM ReactionGame_Optimized
VAR
    // Main button handler
    ButtonHandler : FB_ProcessButtonInput;

    // Helper blocks
    GameOverTrigger : FB_TriggerGameOver;
    NextRoundPrep : FB_PrepareNextRound;

    // Working variables
    NewGapTime : TIME;
END_VAR

// Main LED feedback
OLED_MAIN := NOT IBTN_MAIN;

// Start game
Trig_Start(CLK := IBTN_MAIN AND NOT GameActive AND NOT GameOver_Active);

IF Trig_Start.Q THEN
    GameActive := TRUE;
    Score := 0;
    GapActive := TRUE;
    LEDActive := FALSE;
    CurrentLED := 0;
    T_GameTimer(IN := FALSE, PT := t#60s);
    T_Gap(IN := FALSE);
    T_LED_On(IN := FALSE);

    // Generate first random gap
    Rand_Gen(Execute := TRUE, Seed := 0, Rnd => RandN);
    NewGapTime := F_GetRandomGapTime(RandomValue := RandN);
    T_Gap(PT := NewGapTime);
END_IF;

// Emergency stop
Trig_Mainreset(CLK := IBTN_MAIN AND GameActive AND NOT GameOver_Active);

IF Trig_Mainreset.Q THEN
    GameOverTrigger(
        Execute := TRUE,
        CurrentScore := Score,
        GameActive := GameActive,
        GameOver_Active := GameOver_Active,
        GameOver_Step := GameOver_Step,
        LEDActive := LEDActive,
        GapActive := GapActive,
        HighScore := HighScore
    );

    IF GameOverTrigger.Done THEN
        T_Seq(IN := FALSE, PT := t#300ms);
    END_IF;
ELSE
    GameOverTrigger(Execute := FALSE);
END_IF;

// Main game logic
IF GameActive THEN

    // Run 60 second timer
    T_GameTimer(IN := TRUE, PT := t#60s);

    // Time's up
    IF T_GameTimer.Q THEN
        GameOverTrigger(
            Execute := TRUE,
            CurrentScore := Score,
            GameActive := GameActive,
            GameOver_Active := GameOver_Active,
            GameOver_Step := GameOver_Step,
            LEDActive := LEDActive,
            GapActive := GapActive,
            HighScore := HighScore
        );

        IF GameOverTrigger.Done THEN
            T_Seq(IN := FALSE, PT := t#300ms);
        END_IF;
    END_IF;

    // GAP PHASE
    IF GapActive THEN
        // All LEDs off
        OLED_Y := FALSE;
        OLED_B := FALSE;
        OLED_R := FALSE;
        CurrentLED := 0;

        // Run gap timer
        T_Gap(IN := TRUE);

        // Check button presses
        Trig_Y(CLK := IBTN_Y);
        Trig_B(CLK := IBTN_B);
        Trig_R(CLK := IBTN_R);

        // Process all button inputs with single function block call
        ButtonHandler(
            Yellow_Pressed := Trig_Y.Q,
            Blue_Pressed := Trig_B.Q,
            Red_Pressed := Trig_R.Q,
            CurrentLED := CurrentLED,
            IsGapPhase := TRUE,
            IsLEDPhase := FALSE
        );

        // Handle any button press during gap (all are errors)
        IF ButtonHandler.IsError THEN
            GameOverTrigger(
                Execute := TRUE,
                CurrentScore := Score,
                GameActive := GameActive,
                GameOver_Active := GameOver_Active,
                GameOver_Step := GameOver_Step,
                LEDActive := LEDActive,
                GapActive := GapActive,
                HighScore := HighScore
            );

            T_Seq(IN := FALSE, PT := t#300ms);
            T_Gap(IN := FALSE);
            T_LED_On(IN := FALSE);
        END_IF;

        // Gap finished - light up random LED
        IF T_Gap.Q THEN
            T_Gap(IN := FALSE);
            GapActive := FALSE;
            LEDActive := TRUE;

            Rand_Gen(Execute := TRUE, Seed := 0, Rnd => RandN);
            CurrentLED := F_Rand(RandomValue := RandN);

            // Start 500ms timer
            T_LED_On(IN := FALSE, PT := t#500ms);
        END_IF;
    END_IF;

    // LED PHASE
    IF LEDActive THEN
        // Turn on the appropriate LED
        CASE CurrentLED OF
            1:
                OLED_Y := TRUE;
                OLED_B := FALSE;
                OLED_R := FALSE;
            2:
                OLED_Y := FALSE;
                OLED_B := TRUE;
                OLED_R := FALSE;
            3:
                OLED_Y := FALSE;
                OLED_B := FALSE;
                OLED_R := TRUE;
            ELSE
                OLED_Y := FALSE;
                OLED_B := FALSE;
                OLED_R := FALSE;
        END_CASE;

        // Run LED timer
        T_LED_On(IN := TRUE, PT := t#500ms);

        // Check button presses
        Trig_Y(CLK := IBTN_Y);
        Trig_B(CLK := IBTN_B);
        Trig_R(CLK := IBTN_R);

        // Process all button inputs with single function block call
        ButtonHandler(
            Yellow_Pressed := Trig_Y.Q,
            Blue_Pressed := Trig_B.Q,
            Red_Pressed := Trig_R.Q,
            CurrentLED := CurrentLED,
            IsGapPhase := FALSE,
            IsLEDPhase := TRUE
        );

        // Handle correct button press
        IF ButtonHandler.IsCorrect THEN
            NextRoundPrep(
                Execute := TRUE,
                Score := Score,
                LEDActive := LEDActive,
                GapActive := GapActive
            );

            IF NextRoundPrep.Done THEN
                T_LED_On(IN := FALSE);
                T_Gap(IN := FALSE);
                T_Gap(PT := NextRoundPrep.NewGapTime);
            END_IF;
        ELSE
            NextRoundPrep(Execute := FALSE);
        END_IF;

        // Handle wrong button press
        IF ButtonHandler.IsError THEN
            GameOverTrigger(
                Execute := TRUE,
                CurrentScore := Score,
                GameActive := GameActive,
                GameOver_Active := GameOver_Active,
                GameOver_Step := GameOver_Step,
                LEDActive := LEDActive,
                GapActive := GapActive,
                HighScore := HighScore
            );

            T_Seq(IN := FALSE, PT := t#300ms);
            T_LED_On(IN := FALSE);
            T_Gap(IN := FALSE);
        END_IF;

        // Timer expired - too slow
        IF T_LED_On.Q AND NOT ButtonHandler.IsCorrect THEN
            GameOverTrigger(
                Execute := TRUE,
                CurrentScore := Score,
                GameActive := GameActive,
                GameOver_Active := GameOver_Active,
                GameOver_Step := GameOver_Step,
                LEDActive := LEDActive,
                GapActive := GapActive,
                HighScore := HighScore
            );

            OLED_Y := FALSE;
            OLED_B := FALSE;
            OLED_R := FALSE;

            T_Seq(IN := FALSE, PT := t#300ms);
            T_LED_On(IN := FALSE);
            T_Gap(IN := FALSE);
        END_IF;
    END_IF;
END_IF;

// Game over animation using FB
IF GameOver_Active THEN
    GameOverA(
        Start := TRUE,
        Reset := FALSE
    );

    // Apply LED outputs
    OLED_Y := GameOverA.LED_Yellow;
    OLED_B := GameOverA.LED_Blue;
    OLED_R := GameOverA.LED_Red;

    // Check if animation done
    IF GameOverA.Done THEN
        GameOver_Active := FALSE;
        GameActive := FALSE;
        LEDActive := FALSE;
        GapActive := FALSE;
        Score := 0;
    END_IF;
ELSE
    // Reset animation when not in game over
    GameOverA(
        Start := FALSE,
        Reset := TRUE
    );
END_IF;

END_PROGRAM

(* ---- reaction_game_refactored.st ---- *)
// REFACTORED REACTION GAME LOGIC WITH MODULAR FUNCTIONS

// =============================================================================
// HELPER FUNCTIONS
// =============================================================================

// Function to generate random gap time
FUNCTION F_GenerateRandomGap : TIME
VAR_INPUT
    RandValue : REAL;  // Random value 0.0 to 1.0
END_VAR

IF RandValue < 0.2 THEN
    F_GenerateRandomGap := t#500ms;
ELSIF RandValue < 0.4 THEN
    F_GenerateRandomGap := t#750ms;
ELSIF RandValue < 0.6 THEN
    F_GenerateRandomGap := t#1000ms;
ELSIF RandValue < 0.8 THEN
    F_GenerateRandomGap := t#1250ms;
ELSE
    F_GenerateRandomGap := t#1500ms;
END_IF;

END_FUNCTION

// =============================================================================
// FUNCTION BLOCK FOR BUTTON PRESS HANDLING
// =============================================================================

FUNCTION_BLOCK FB_HandleButtonPress
VAR_INPUT
    ButtonPressed : BOOL;      // Trigger from button press
    ButtonID : INT;           // Which button (1=Yellow, 2=Blue, 3=Red)
    CurrentLED : INT;          // Which LED is currently on
    GamePhase : INT;           // 0=Gap, 1=LED Active
END_VAR

VAR_OUTPUT
    CorrectPress : BOOL;       // TRUE if correct button pressed
    WrongPress : BOOL;         // TRUE if wrong button/timing
    UpdateScore : BOOL;        // TRUE to increment score
END_VAR

VAR
    // Internal processing
END_VAR

// Reset outputs
CorrectPress := FALSE;
WrongPress := FALSE;
UpdateScore := FALSE;

IF ButtonPressed THEN
    IF GamePhase = 0 THEN
        // Button pressed during gap phase - always wrong
        WrongPress := TRUE;
    ELSIF GamePhase = 1 THEN
        // Button pressed during LED phase
        IF ButtonID = CurrentLED THEN
            // Correct button!
            CorrectPress := TRUE;
            UpdateScore := TRUE;
        ELSE
            // Wrong button
            WrongPress := TRUE;
        END_IF;
    END_IF;
END_IF;

END_FUNCTION_BLOCK

// =============================================================================
// FUNCTION BLOCK FOR GAME OVER SEQUENCE
// =============================================================================

FUNCTION_BLOCK FB_InitGameOver
VAR_INPUT
    Trigger : BOOL;            // Trigger to start game over
    CurrentScore : INT;        // Current game score
END_VAR

VAR_IN_OUT
    HighScore : INT;           // High score to update
    GameActive : BOOL;         // Game active flag
    GameOver_Active : BOOL;    // Game over flag
    GameOver_Step : INT;       // Game over animation step
    LEDActive : BOOL;          // LED phase flag
    GapActive : BOOL;          // Gap phase flag
END_VAR

VAR_OUTPUT
    // Timers to reset
    ResetTimers : BOOL;
END_VAR

IF Trigger THEN
    // Set game over state
    GameActive := FALSE;
    GameOver_Active := TRUE;
    GameOver_Step := 0;
    LEDActive := FALSE;
    GapActive := FALSE;
    ResetTimers := TRUE;

    // Update high score if needed
    IF CurrentScore > HighScore THEN
        HighScore := CurrentScore;
    END_IF;
ELSE
    ResetTimers := FALSE;
END_IF;

END_FUNCTION_BLOCK

// =============================================================================
// MAIN PROGRAM - REFACTORED
// =============================================================================

PROGRAM ReactionGame_Main
VAR
    // Button handlers
    ButtonHandler_Y : FB_HandleButtonPress;
    ButtonHandler_B : FB_HandleButtonPress;
    ButtonHandler_R : FB_HandleButtonPress;

    // Game over handler
    GameOverHandler : FB_InitGameOver;

    // Temporary variables for button processing
    ButtonProcessed : BOOL;
    NextGapTime : TIME;
END_VAR

// MAIN Logic reaction game

// Main LED feedback
OLED_MAIN := NOT IBTN_MAIN;

// Start game
Trig_Start(CLK := IBTN_MAIN AND NOT GameActive AND NOT GameOver_Active);

IF Trig_Start.Q THEN
    GameActive := TRUE;
    Score := 0;
    GapActive := TRUE;
    LEDActive := FALSE;
    CurrentLED := 0;
    T_GameTimer(IN := FALSE, PT := t#60s);
    T_Gap(IN := FALSE);
    T_LED_On(IN := FALSE);

    // Generate first random gap
    Rand_Gen(Execute := TRUE, Seed := 0, Rnd => RandN);
    NextGapTime := F_GenerateRandomGap(RandValue := RandN);
    T_Gap(PT := NextGapTime);
END_IF;

// Emergency stop
Trig_Mainreset(CLK := IBTN_MAIN AND GameActive AND NOT GameOver_Active);

IF Trig_Mainreset.Q THEN
    GameOverHandler(
        Trigger := TRUE,
        CurrentScore := Score,
        HighScore := HighScore,
        GameActive := GameActive,
        GameOver_Active := GameOver_Active,
        GameOver_Step := GameOver_Step,
        LEDActive := LEDActive,
        GapActive := GapActive
    );

    IF GameOverHandler.ResetTimers THEN
        T_Seq(IN := FALSE, PT := t#300ms);
        T_Gap(IN := FALSE);
        T_LED_On(IN := FALSE);
    END_IF;
ELSE
    GameOverHandler(Trigger := FALSE);
END_IF;

// Main game logic
IF GameActive THEN

    // Run 60 second timer
    T_GameTimer(IN := TRUE, PT := t#60s);

    // Time's up
    IF T_GameTimer.Q THEN
        GameOverHandler(
            Trigger := TRUE,
            CurrentScore := Score,
            HighScore := HighScore,
            GameActive := GameActive,
            GameOver_Active := GameOver_Active,
            GameOver_Step := GameOver_Step,
            LEDActive := LEDActive,
            GapActive := GapActive
        );

        IF GameOverHandler.ResetTimers THEN
            T_Seq(IN := FALSE, PT := t#300ms);
        END_IF;
    END_IF;

    // Determine current game phase (0=Gap, 1=LED Active)
    VAR
        CurrentPhase : INT;
    END_VAR

    IF GapActive THEN
        CurrentPhase := 0;
    ELSIF LEDActive THEN
        CurrentPhase := 1;
    ELSE
        CurrentPhase := -1;
    END_IF;

    // GAP PHASE - waiting for LED (don't press anything!)
    IF GapActive THEN
        // All LEDs off
        OLED_Y := FALSE;
        OLED_B := FALSE;
        OLED_R := FALSE;
        CurrentLED := 0;

        // Run gap timer
        T_Gap(IN := TRUE);

        // Check for button presses using function blocks
        Trig_Y(CLK := IBTN_Y);
        Trig_B(CLK := IBTN_B);
        Trig_R(CLK := IBTN_R);

        ButtonProcessed := FALSE;

        // Handle Yellow button
        ButtonHandler_Y(
            ButtonPressed := Trig_Y.Q,
            ButtonID := 1,
            CurrentLED := CurrentLED,
            GamePhase := CurrentPhase
        );

        // Handle Blue button
        ButtonHandler_B(
            ButtonPressed := Trig_B.Q,
            ButtonID := 2,
            CurrentLED := CurrentLED,
            GamePhase := CurrentPhase
        );

        // Handle Red button
        ButtonHandler_R(
            ButtonPressed := Trig_R.Q,
            ButtonID := 3,
            CurrentLED := CurrentLED,
            GamePhase := CurrentPhase
        );

        // Any wrong press during gap = game over
        IF ButtonHandler_Y.WrongPress OR ButtonHandler_B.WrongPress OR ButtonHandler_R.WrongPress THEN
            GameOverHandler(
                Trigger := TRUE,
                CurrentScore := Score,
                HighScore := HighScore,
                GameActive := GameActive,
                GameOver_Active := GameOver_Active,
                GameOver_Step := GameOver_Step,
                LEDActive := LEDActive,
                GapActive := GapActive
            );

            IF GameOverHandler.ResetTimers THEN
                T_Seq(IN := FALSE, PT := t#300ms);
                T_Gap(IN := FALSE);
                T_LED_On(IN := FALSE);
            END_IF;
        END_IF;

        // Gap finished - light up random LED
        IF T_Gap.Q THEN
            T_Gap(IN := FALSE);
            GapActive := FALSE;
            LEDActive := TRUE;

            Rand_Gen(Execute := TRUE, Seed := 0, Rnd => RandN);
            CurrentLED := F_Rand(RandomValue := RandN);

            // Start 500ms timer
            T_LED_On(IN := FALSE, PT := t#500ms);
        END_IF;
    END_IF;

    // LED PHASE - press the correct button
    IF LEDActive THEN
        // Turn on the LED
        CASE CurrentLED OF
            1: OLED_Y := TRUE; OLED_B := FALSE; OLED_R := FALSE;
            2: OLED_Y := FALSE; OLED_B := TRUE; OLED_R := FALSE;
            3: OLED_Y := FALSE; OLED_B := FALSE; OLED_R := TRUE;
            ELSE OLED_Y := FALSE; OLED_B := FALSE; OLED_R := FALSE;
        END_CASE;

        // Run LED timer
        T_LED_On(IN := TRUE, PT := t#500ms);

        // Check button presses
        Trig_Y(CLK := IBTN_Y);
        Trig_B(CLK := IBTN_B);
        Trig_R(CLK := IBTN_R);

        ButtonProcessed := FALSE;

        // Handle Yellow button
        ButtonHandler_Y(
            ButtonPressed := Trig_Y.Q,
            ButtonID := 1,
            CurrentLED := CurrentLED,
            GamePhase := CurrentPhase
        );

        // Handle Blue button
        ButtonHandler_B(
            ButtonPressed := Trig_B.Q,
            ButtonID := 2,
            CurrentLED := CurrentLED,
            GamePhase := CurrentPhase
        );

        // Handle Red button
        ButtonHandler_R(
            ButtonPressed := Trig_R.Q,
            ButtonID := 3,
            CurrentLED := CurrentLED,
            GamePhase := CurrentPhase
        );

        // Process button results (only one can be pressed at a time)
        IF ButtonHandler_Y.CorrectPress OR ButtonHandler_B.CorrectPress OR ButtonHandler_R.CorrectPress THEN
            // Correct button pressed
            Score := Score + 1;
            LEDActive := FALSE;
            GapActive := TRUE;
            T_LED_On(IN := FALSE);

            // Generate next random gap
            Rand_Gen(Execute := TRUE, Seed := 0, Rnd => RandN);
            NextGapTime := F_GenerateRandomGap(RandValue := RandN);
            T_Gap(IN := FALSE);
            T_Gap(PT := NextGapTime);

            ButtonProcessed := TRUE;
        ELSIF ButtonHandler_Y.WrongPress OR ButtonHandler_B.WrongPress OR ButtonHandler_R.WrongPress THEN
            // Wrong button pressed
            GameOverHandler(
                Trigger := TRUE,
                CurrentScore := Score,
                HighScore := HighScore,
                GameActive := GameActive,
                GameOver_Active := GameOver_Active,
                GameOver_Step := GameOver_Step,
                LEDActive := LEDActive,
                GapActive := GapActive
            );

            IF GameOverHandler.ResetTimers THEN
                T_Seq(IN := FALSE, PT := t#300ms);
                T_LED_On(IN := FALSE);
                T_Gap(IN := FALSE);
            END_IF;

            ButtonProcessed := TRUE;
        END_IF;

        // Timer expired - too slow
        IF T_LED_On.Q AND NOT ButtonProcessed THEN
            GameOverHandler(
                Trigger := TRUE,
                CurrentScore := Score,
                HighScore := HighScore,
                GameActive := GameActive,
                GameOver_Active := GameOver_Active,
                GameOver_Step := GameOver_Step,
                LEDActive := LEDActive,
                GapActive := GapActive
            );

            OLED_Y := FALSE;
            OLED_B := FALSE;
            OLED_R := FALSE;

            IF GameOverHandler.ResetTimers THEN
                T_Seq(IN := FALSE, PT := t#300ms);
                T_LED_On(IN := FALSE);
                T_Gap(IN := FALSE);
            END_IF;
        END_IF;
    END_IF;
END_IF;

// Game over animation using FB
IF GameOver_Active THEN
    GameOverA(
        Start := TRUE,
        Reset := FALSE
    );

    // Apply LED outputs
    OLED_Y := GameOverA.LED_Yellow;
    OLED_B := GameOverA.LED_Blue;
    OLED_R := GameOverA.LED_Red;

    // Check if animation done
    IF GameOverA.Done THEN
        GameOver_Active := FALSE;
        GameActive := FALSE;
        LEDActive := FALSE;
        GapActive := FALSE;
        Score := 0;
    END_IF;
ELSE
    // Reset animation when not in game over
    GameOverA(
        Start := FALSE,
        Reset := TRUE
    );
END_IF;

END_PROGRAM

(* ---- simon_says_timer_functions.st ---- *)
(* Simon Says Game - Timer Functions and Utilities *)
(* For Omron NX102-1100 PLC *)

(* ============================================================================ *)
(* FUNCTION BLOCK: SequenceTimer *)
(* Purpose: Manages timing for sequence display with adjustable flash and gap times *)
(* ============================================================================ *)

FUNCTION_BLOCK SequenceTimer
VAR_INPUT
    Enable      : BOOL;     (* Enable the timer *)
    FlashTime   : TIME;     (* Duration for LED flash *)
    GapTime     : TIME;     (* Duration for gap between flashes *)
    Reset       : BOOL;     (* Reset the timer *)
END_VAR

VAR_OUTPUT
    FlashActive : BOOL;     (* TRUE when LED should be on *)
    StepComplete: BOOL;     (* TRUE when one complete flash+gap cycle is done *)
    Busy        : BOOL;     (* TRUE when timer is running *)
END_VAR

VAR
    FlashTimer  : TON;      (* Timer for flash duration *)
    GapTimer    : TON;      (* Timer for gap duration *)
    State       : INT;      (* 0=Idle, 1=Flash, 2=Gap *)
END_VAR

(* Reset logic *)
IF Reset THEN
    State := 0;
    FlashActive := FALSE;
    StepComplete := FALSE;
    Busy := FALSE;
    FlashTimer(IN := FALSE);
    GapTimer(IN := FALSE);
    RETURN;
END_IF;

(* Main timer logic *)
IF Enable THEN
    Busy := TRUE;

    CASE State OF
        0: (* Idle - start flash *)
            IF Enable THEN
                State := 1;
                FlashActive := TRUE;
                StepComplete := FALSE;
            END_IF;

        1: (* Flash phase *)
            FlashTimer(IN := TRUE, PT := FlashTime);
            IF FlashTimer.Q THEN
                FlashActive := FALSE;
                State := 2;
                FlashTimer(IN := FALSE);
            END_IF;

        2: (* Gap phase *)
            GapTimer(IN := TRUE, PT := GapTime);
            IF GapTimer.Q THEN
                StepComplete := TRUE;
                State := 0;
                GapTimer(IN := FALSE);
                Busy := FALSE;
            END_IF;
    END_CASE;
ELSE
    Busy := FALSE;
    FlashActive := FALSE;
    StepComplete := FALSE;
    State := 0;
END_IF;

END_FUNCTION_BLOCK

(* ============================================================================ *)
(* FUNCTION BLOCK: InputTimer *)
(* Purpose: Manages player input timeout with visual countdown *)
(* ============================================================================ *)

FUNCTION_BLOCK InputTimer
VAR_INPUT
    Enable      : BOOL;     (* Start the input timer *)
    TimeoutValue: TIME;     (* Timeout duration *)
    Reset       : BOOL;     (* Reset the timer *)
END_VAR

VAR_OUTPUT
    TimeExpired : BOOL;     (* TRUE when timeout occurs *)
    TimeRemaining: TIME;    (* Time remaining *)
    WarningActive: BOOL;    (* TRUE when in warning period (last 25% of time) *)
END_VAR

VAR
    InputTimer  : TON;      (* Main timeout timer *)
    ElapsedTime : TIME;     (* Elapsed time *)
END_VAR

(* Reset logic *)
IF Reset THEN
    TimeExpired := FALSE;
    TimeRemaining := TimeoutValue;
    WarningActive := FALSE;
    InputTimer(IN := FALSE);
    RETURN;
END_IF;

(* Timer logic *)
InputTimer(IN := Enable, PT := TimeoutValue);

IF Enable THEN
    ElapsedTime := InputTimer.ET;
    TimeRemaining := TimeoutValue - ElapsedTime;

    (* Warning when 75% of time has elapsed *)
    WarningActive := (ElapsedTime >= (TimeoutValue * 3 / 4));

    (* Timeout check *)
    TimeExpired := InputTimer.Q;
ELSE
    TimeRemaining := TimeoutValue;
    WarningActive := FALSE;
    TimeExpired := FALSE;
END_IF;

END_FUNCTION_BLOCK

(* ============================================================================ *)
(* FUNCTION BLOCK: CelebrationTimer *)
(* Purpose: Manages success celebration effects *)
(* ============================================================================ *)

FUNCTION_BLOCK CelebrationTimer
VAR_INPUT
    Trigger     : BOOL;     (* Start celebration *)
    Duration    : TIME;     (* Celebration duration *)
END_VAR

VAR_OUTPUT
    Active      : BOOL;     (* TRUE during celebration *)
    FlashPattern: BOOL;     (* Flashing pattern for LEDs *)
    Complete    : BOOL;     (* TRUE when celebration is finished *)
END_VAR

VAR
    CelebTimer  : TON;      (* Main celebration timer *)
    FlashTimer  : TON;      (* Flash pattern timer *)
    TriggerEdge : R_TRIG;   (* Edge detection for trigger *)
END_VAR

TriggerEdge(CLK := Trigger);

IF TriggerEdge.Q THEN
    Active := TRUE;
    Complete := FALSE;
    CelebTimer(IN := FALSE); (* Reset timer *)
END_IF;

IF Active THEN
    CelebTimer(IN := TRUE, PT := Duration);

    (* Create flash pattern (200ms on/off) *)
    FlashTimer(IN := TRUE, PT := T#200ms);
    IF FlashTimer.Q THEN
        FlashPattern := NOT FlashPattern;
        FlashTimer(IN := FALSE);
    END_IF;

    (* Check if celebration is complete *)
    IF CelebTimer.Q THEN
        Active := FALSE;
        Complete := TRUE;
        FlashPattern := FALSE;
    END_IF;
ELSE
    FlashPattern := FALSE;
    IF Complete THEN
        Complete := FALSE; (* Reset complete flag after one scan *)
    END_IF;
END_IF;

END_FUNCTION_BLOCK

(* ============================================================================ *)
(* FUNCTION BLOCK: ErrorTimer *)
(* Purpose: Manages game over error display *)
(* ============================================================================ *)

FUNCTION_BLOCK ErrorTimer
VAR_INPUT
    Trigger     : BOOL;     (* Start error display *)
    BlinkCount  : INT;      (* Number of blinks (default 3) *)
    BlinkSpeed  : TIME;     (* Blink speed (default 200ms) *)
    HoldTime    : TIME;     (* Final hold time (default 2s) *)
END_VAR

VAR_OUTPUT
    Active      : BOOL;     (* TRUE during error display *)
    BlinkState  : BOOL;     (* Blink pattern for LEDs *)
    Complete    : BOOL;     (* TRUE when error display is finished *)
END_VAR

VAR
    BlinkTimer  : TON;      (* Blink timing *)
    HoldTimer   : TON;      (* Final hold timing *)
    TriggerEdge : R_TRIG;   (* Edge detection *)
    BlinkCounter: INT;      (* Current blink count *)
    Phase       : INT;      (* 0=Blink, 1=Hold *)
END_VAR

TriggerEdge(CLK := Trigger);

IF TriggerEdge.Q THEN
    Active := TRUE;
    Complete := FALSE;
    BlinkCounter := 0;
    Phase := 0;
    BlinkState := FALSE;
    BlinkTimer(IN := FALSE);
    HoldTimer(IN := FALSE);
END_IF;

IF Active THEN
    CASE Phase OF
        0: (* Blinking phase *)
            BlinkTimer(IN := TRUE, PT := BlinkSpeed);
            IF BlinkTimer.Q THEN
                BlinkState := NOT BlinkState;
                BlinkCounter := BlinkCounter + 1;
                BlinkTimer(IN := FALSE);

                IF BlinkCounter >= (BlinkCount * 2) THEN (* *2 for on/off cycles *)
                    Phase := 1;
                    BlinkState := TRUE; (* Final state ON *)
                END_IF;
            END_IF;

        1: (* Hold phase *)
            HoldTimer(IN := TRUE, PT := HoldTime);
            IF HoldTimer.Q THEN
                Active := FALSE;
                Complete := TRUE;
                BlinkState := FALSE;
            END_IF;
    END_CASE;
ELSE
    BlinkState := FALSE;
    IF Complete THEN
        Complete := FALSE; (* Reset complete flag *)
    END_IF;
END_IF;

END_FUNCTION_BLOCK

(* ============================================================================ *)
(* FUNCTION: RandomGenerator *)
(* Purpose: Generate random numbers for sequence *)
(* ============================================================================ *)

FUNCTION RandomGenerator : INT
VAR_INPUT
    Seed        : DINT;     (* Random seed *)
    MinValue    : INT;      (* Minimum value (inclusive) *)
    MaxValue    : INT;      (* Maximum value (inclusive) *)
END_VAR

VAR
    NewSeed     : DINT;
    Range       : INT;
END_VAR

(* Linear Congruential Generator *)
NewSeed := Seed * 1103515245 + 12345;

(* Calculate range *)
Range := MaxValue - MinValue + 1;

(* Return random value in range *)
RandomGenerator := MinValue + (NewSeed MOD Range);

END_FUNCTION

(* ============================================================================ *)
(* FUNCTION BLOCK: GameDifficulty *)
(* Purpose: Manages difficulty settings for future phases *)
(* ============================================================================ *)

FUNCTION_BLOCK GameDifficulty
VAR_INPUT
    DifficultyLevel : INT;  (* 0=Easy, 1=Normal, 2=Hard *)
END_VAR

VAR_OUTPUT
    FlashTime       : TIME; (* LED flash duration *)
    GapTime         : TIME; (* Gap between flashes *)
    InputTimeout    : TIME; (* Player input timeout *)
    MaxSequence     : INT;  (* Maximum sequence length *)
END_VAR

CASE DifficultyLevel OF
    0: (* Easy *)
        FlashTime := T#800ms;
        GapTime := T#400ms;
        InputTimeout := T#5s;
        MaxSequence := 10;

    1: (* Normal *)
        FlashTime := T#500ms;
        GapTime := T#200ms;
        InputTimeout := T#3s;
        MaxSequence := 15;

    2: (* Hard *)
        FlashTime := T#300ms;
        GapTime := T#100ms;
        InputTimeout := T#2s;
        MaxSequence := 20;

    ELSE (* Default to Normal *)
        FlashTime := T#500ms;
        GapTime := T#200ms;
        InputTimeout := T#3s;
        MaxSequence := 15;
END_CASE;

END_FUNCTION_BLOCK

(* ---- GameFlow_Logic.st ---- *)
PROGRAM GameFlow_Logic
VAR
    // Existing variables
    B : BOOL;                    // Button trigger
    RandN : REAL;                // Random number 0.0-1.0
    L_N : INT;                   // LED number (1-3)
    WriteIndex : LINT := 0;      // Array write index
    Idx : INT;                   // Converted index for array access
    ArrayFull : BOOL := FALSE;   // Array full flag

    // Array declarations
    GameFlow_S : ARRAY[0..49] OF INT;     // Source array
    GameFlow_SN : ARRAY[0..49] OF INT;    // New array for reset

    // Reset signal handling
    ResetSignal : BOOL;          // Reset signal input
    ResetTrigger : BOOL;         // Rising edge detection for reset

    // LED control variables
    OLED_R : BOOL;               // Red LED
    OLED_B : BOOL;               // Blue LED
    OLED_Y : BOOL;               // Yellow LED

    // Game over sequence variables
    GameOverActive : BOOL := FALSE;
    GameOverTimer : TIME := T#0s;
    GameOverStep : INT := 0;
    GameOverStepTime : TIME := T#1s;  // 1 second per step

    // LED sequence pattern (1=Red, 2=Blue, 3=Yellow)
    LEDSequence : ARRAY[0..8] OF INT := [1, 2, 3, 1, 2, 3, 1, 2, 3];
    SequenceIndex : INT := 0;

END_VAR

// Rising edge detection for button
Trig_Start(Clk := IBTN_B, Q => B);

// Rising edge detection for reset signal
Trig_Start(Clk := ResetSignal, Q => ResetTrigger);

// Reset signal handling
IF ResetTrigger THEN
    // Add current game flow to array when reset is triggered
    AryAddV(In1 := GameFlow_S[0], In2 := L_N, Size := 50, AryOut := GameFlow_SN[0]);

    // Start game over sequence
    GameOverActive := TRUE;
    GameOverTimer := T#0s;
    GameOverStep := 0;
    SequenceIndex := 0;
END_IF;

// Game over LED sequence
IF GameOverActive THEN
    GameOverTimer := GameOverTimer + T#10ms;  // Increment timer (assuming 10ms cycle)

    // Check if it's time for next step
    IF GameOverTimer >= GameOverStepTime THEN
        GameOverTimer := T#0s;
        GameOverStep := GameOverStep + 1;

        // Turn off all LEDs
        OLED_R := FALSE;
        OLED_B := FALSE;
        OLED_Y := FALSE;

        // Check if sequence is complete
        IF GameOverStep >= 9 THEN  // 9 steps total (3 cycles of 3 LEDs)
            GameOverActive := FALSE;
            GameOverStep := 0;
            SequenceIndex := 0;
        ELSE
            // Light up the appropriate LED based on sequence
            CASE LEDSequence[SequenceIndex] OF
                1: OLED_R := TRUE;   // Red LED
                2: OLED_B := TRUE;   // Blue LED
                3: OLED_Y := TRUE;   // Yellow LED
            END_CASE;

            SequenceIndex := SequenceIndex + 1;
        END_IF;
    END_IF;
END_IF;

// Original button press logic (only when not in game over sequence)
IF B AND NOT GameOverActive THEN
    // Random number 0.0–1.0
    Rand_Gen(Execute := TRUE, Seed := 0, Rnd => RandN);

    // Map to 1..3
    IF RandN < 0.333 THEN
        L_N := 1;
    ELSIF RandN < 0.666 THEN
        L_N := 2;
    ELSE
        L_N := 3;
    END_IF;

    // Keep WriteIndex in 0..49 and set "full" once we wrap
    IF WriteIndex >= 50 THEN
        WriteIndex := 0;
        ArrayFull := TRUE;
    ELSIF WriteIndex < 0 THEN
        // (safety, in case WriteIndex ever goes negative)
        WriteIndex := 0;
    END_IF;

    // Convert LINT -> INT for array subscript
    Idx := TO_INT(WriteIndex);          // or: Idx := LINT_TO_INT(WriteIndex);

    // Write value into the next slot
    GameFlow_SN[Idx] := L_N;
    // Optional mirror:
    // GameFlow_S[Idx] := L_N;

    // Advance for next press
    WriteIndex := WriteIndex + 1;
END_IF;

END_PROGRAM

(* ---- MAIN_ReactionGame_Refactored.st ---- *)
// MAIN Logic reaction game (REFACTORED)

VAR
    // Function block instances for button checking
    CheckYellow : FB_CheckButtonPress;
    CheckBlue : FB_CheckButtonPress;
    CheckRed : FB_CheckButtonPress;

    // Other variables (your existing declarations)
    // ... add your other VAR declarations here
END_VAR

// Main LED feedback
OLED_MAIN := NOT IBTN_MAIN;

// Start game
Trig_Start(CLK := IBTN_MAIN AND NOT GameActive AND NOT GameOver_Active);

IF Trig_Start.Q THEN
    GameActive := TRUE;
    Score := 0;
    GapActive := TRUE;
    LEDActive := FALSE;
    CurrentLED := 0;
    T_GameTimer(IN := FALSE, PT := t#60s);
    T_Gap(IN := FALSE);
    T_LED_On(IN := FALSE);

    // Generate first random gap
    Rand_Gen(Execute := TRUE, Seed := 0, Rnd => RandN);
    IF RandN < 0.2 THEN
        T_Gap(PT := t#500ms);
    ELSIF RandN < 0.4 THEN
        T_Gap(PT := t#750ms);
    ELSIF RandN < 0.6 THEN
        T_Gap(PT := t#1000ms);
    ELSIF RandN < 0.8 THEN
        T_Gap(PT := t#1250ms);
    ELSE
        T_Gap(PT := t#1500ms);
    END_IF;
END_IF;

// Emergency stop
Trig_Mainreset(CLK := IBTN_MAIN AND GameActive AND NOT GameOver_Active);

IF Trig_Mainreset.Q THEN
    GameActive := FALSE;
    GameOver_Active := TRUE;
    GameOver_Step := 0;
    T_Seq(IN := FALSE, PT := t#300ms);
END_IF;

// Main game logic
IF GameActive THEN

    // Run 60 second timer
    T_GameTimer(IN := TRUE, PT := t#60s);

    // Time's up
    IF T_GameTimer.Q THEN
        GameActive := FALSE;
        GameOver_Active := TRUE;
        GameOver_Step := 0;
        T_Seq(IN := FALSE, PT := t#300ms);

        IF Score > HighScore THEN
            HighScore := Score;
        END_IF;
    END_IF;

    // GAP PHASE - waiting for LED (don't press anything!)
    IF GapActive THEN
        // All LEDs off
        OLED_Y := FALSE;
        OLED_B := FALSE;
        OLED_R := FALSE;
        CurrentLED := 0;

        // Run gap timer
        T_Gap(IN := TRUE);

        // Check for early button press
        Trig_Y(CLK := IBTN_Y);
        Trig_B(CLK := IBTN_B);
        Trig_R(CLK := IBTN_R);

        // Pressed during gap - instant game over
        IF Trig_Y.Q OR Trig_B.Q OR Trig_R.Q THEN
            GameActive := FALSE;
            GameOver_Active := TRUE;
            GameOver_Step := 0;
            T_Seq(IN := FALSE, PT := t#300ms);
            GapActive := FALSE;
            LEDActive := FALSE;
            T_Gap(IN := FALSE);
            T_LED_On(IN := FALSE);

            IF Score > HighScore THEN
                HighScore := Score;
            END_IF;
        END_IF;

        // Gap finished - light up random LED
        IF T_Gap.Q THEN
            T_Gap(IN := FALSE);
            GapActive := FALSE;
            LEDActive := TRUE;

            Rand_Gen(Execute := TRUE, Seed := 0, Rnd => RandN);
            CurrentLED := F_Rand(RandomValue := RandN);

            // Start 500ms timer
            T_LED_On(IN := FALSE, PT := t#500ms);
        END_IF;
    END_IF;

    // LED PHASE - press the correct button
    IF LEDActive THEN
        // Turn on the LED
        CASE CurrentLED OF
            1: OLED_Y := TRUE; OLED_B := FALSE; OLED_R := FALSE;
            2: OLED_Y := FALSE; OLED_B := TRUE; OLED_R := FALSE;
            3: OLED_Y := FALSE; OLED_B := FALSE; OLED_R := TRUE;
            ELSE OLED_Y := FALSE; OLED_B := FALSE; OLED_R := FALSE;
        END_CASE;

        // Run LED timer
        T_LED_On(IN := TRUE, PT := t#500ms);

        // Check button presses
        Trig_Y(CLK := IBTN_Y);
        Trig_B(CLK := IBTN_B);
        Trig_R(CLK := IBTN_R);

        // ====== REFACTORED BUTTON CHECKING ======
        // Check Yellow button
        CheckYellow(
            ButtonPressed := Trig_Y.Q,
            ExpectedLED := 1,
            CurrentLED := CurrentLED,
            Score := Score,
            HighScore := HighScore
        );

        // Check Blue button
        CheckBlue(
            ButtonPressed := Trig_B.Q,
            ExpectedLED := 2,
            CurrentLED := CurrentLED,
            Score := Score,
            HighScore := HighScore
        );

        // Check Red button
        CheckRed(
            ButtonPressed := Trig_R.Q,
            ExpectedLED := 3,
            CurrentLED := CurrentLED,
            Score := Score,
            HighScore := HighScore
        );

        // Handle correct button press (any of the three)
        IF CheckYellow.ContinueGame OR CheckBlue.ContinueGame OR CheckRed.ContinueGame THEN
            // Update score
            IF CheckYellow.ContinueGame THEN
                Score := CheckYellow.NewScore;
                T_Gap(PT := CheckYellow.NextGapTime);
            ELSIF CheckBlue.ContinueGame THEN
                Score := CheckBlue.NewScore;
                T_Gap(PT := CheckBlue.NextGapTime);
            ELSIF CheckRed.ContinueGame THEN
                Score := CheckRed.NewScore;
                T_Gap(PT := CheckRed.NextGapTime);
            END_IF;

            // Continue to next round
            LEDActive := FALSE;
            GapActive := TRUE;
            T_LED_On(IN := FALSE);
            T_Gap(IN := FALSE);
        END_IF;

        // Handle wrong button press (game over)
        IF CheckYellow.EndGame OR CheckBlue.EndGame OR CheckRed.EndGame THEN
            // Update high score
            IF CheckYellow.EndGame THEN
                HighScore := CheckYellow.NewHighScore;
            ELSIF CheckBlue.EndGame THEN
                HighScore := CheckBlue.NewHighScore;
            ELSIF CheckRed.EndGame THEN
                HighScore := CheckRed.NewHighScore;
            END_IF;

            // End game
            GameActive := FALSE;
            GameOver_Active := TRUE;
            GameOver_Step := 0;
            T_Seq(IN := FALSE, PT := t#300ms);
            LEDActive := FALSE;
            GapActive := FALSE;
            T_LED_On(IN := FALSE);
            T_Gap(IN := FALSE);
        END_IF;
        // ====== END REFACTORED SECTION ======

        // Timer expired - too slow
        IF T_LED_On.Q THEN
            GameActive := FALSE;
            GameOver_Active := TRUE;
            GameOver_Step := 0;
            T_Seq(IN := FALSE, PT := t#300ms);
            LEDActive := FALSE;
            GapActive := FALSE;
            OLED_Y := FALSE;
            OLED_B := FALSE;
            OLED_R := FALSE;
            T_LED_On(IN := FALSE);
            T_Gap(IN := FALSE);

            IF Score > HighScore THEN
                HighScore := Score;
            END_IF;
        END_IF;
    END_IF;
END_IF;

// Game over animation using FB
IF GameOver_Active THEN
    GameOverA(
        Start := TRUE,
        Reset := FALSE
    );

    // Apply LED outputs
    OLED_Y := GameOverA.LED_Yellow;
    OLED_B := GameOverA.LED_Blue;
    OLED_R := GameOverA.LED_Red;

    // Check if animation done
    IF GameOverA.Done THEN
        GameOver_Active := FALSE;
        GameActive := FALSE;
        LEDActive := FALSE;
        GapActive := FALSE;
        Score := 0;
    END_IF;
ELSE
    // Reset animation when not in game over
    GameOverA(
        Start := FALSE,
        Reset := TRUE
    );
END_IF;

(* ---- MainProgram.st ---- *)
(* ====================================================================== *)
(* Main Program - Simon Says Game                                        *)
(* Uses FB_SimonSays Function Block                                      *)
(* For Omron NX102-1100 PLC                                             *)
(* ====================================================================== *)

PROGRAM MainProgram

VAR_GLOBAL
    (* ====================================================================== *)
    (* Physical I/O Mapping                                                  *)
    (* ====================================================================== *)
    (* Inputs from NX-ID4442 *)
    DI_YellowButton AT %IX0.1 : BOOL;    (* DI1 - Yellow button contact *)
    DI_BlueButton AT %IX0.3 : BOOL;      (* DI3 - Blue button contact *)
    DI_RedButton AT %IX0.5 : BOOL;       (* DI5 - Red button contact *)

    (* Outputs to NX-OD4256 *)
    DO_RedLED AT %QX0.0 : BOOL;          (* DO0 - Red button LED *)
    DO_BlueLED AT %QX0.1 : BOOL;         (* DO1 - Blue button LED *)
    DO_YellowLED AT %QX0.2 : BOOL;       (* DO2 - Yellow button LED *)

    (* Control Inputs - Map to selector switch later *)
    StartButton : BOOL := FALSE;          (* Start game signal *)
    ResetButton : BOOL := FALSE;          (* Reset game signal *)

    (* Game Instance *)
    SimonSaysGame : FB_SimonSays;

    (* HMI Variables *)
    GameActive : BOOL;
    CurrentLevel : INT;
    GameWon : BOOL;
    GameLost : BOOL;
    CurrentState : INT;

    (* Configuration Parameters *)
    MaxLevel : INT := 10;                 (* Maximum sequence length *)
    ShowTime : TIME := T#500MS;           (* LED display duration *)
    GapTime : TIME := T#200MS;            (* Gap between LEDs *)
    InputTimeout : TIME := T#3S;          (* Player input timeout *)

END_VAR

(* ====================================================================== *)
(* MAIN PROGRAM EXECUTION                                                *)
(* ====================================================================== *)

(* Call Simon Says Function Block *)
SimonSaysGame(
    (* Inputs *)
    i_YellowButton := DI_YellowButton,
    i_BlueButton := DI_BlueButton,
    i_RedButton := DI_RedButton,
    i_StartButton := StartButton,
    i_Reset := ResetButton,
    i_MaxLevel := MaxLevel,
    i_ShowTime := ShowTime,
    i_GapTime := GapTime,
    i_InputTimeout := InputTimeout,

    (* Outputs *)
    q_YellowLED => DO_YellowLED,
    q_BlueLED => DO_BlueLED,
    q_RedLED => DO_RedLED,
    q_GameActive => GameActive,
    q_CurrentLevel => CurrentLevel,
    q_GameWon => GameWon,
    q_GameLost => GameLost,
    q_State => CurrentState
);

(* ====================================================================== *)
(* Additional Logic for Selector Switch Integration                      *)
(* Map selector switch positions to game control                         *)
(* This will be expanded in Phase 2                                      *)
(* ====================================================================== *)

(* For now, you can manually set StartButton to TRUE to start the game *)
(* In actual implementation, this would be connected to selector switch *)

END_PROGRAM

(* ---- ReactionGameMain_Refactored.st ---- *)
// MAIN Logic reaction game

// Main LED feedback
OLED_MAIN := NOT IBTN_MAIN;

// Start game
Trig_Start(CLK := IBTN_MAIN AND NOT GameActive AND NOT GameOver_Active);

IF Trig_Start.Q THEN
    GameActive := TRUE;
    Score := 0;
    GapActive := TRUE;
    LEDActive := FALSE;
    CurrentLED := 0;
    T_GameTimer(IN := FALSE, PT := t#60s);
    T_Gap(IN := FALSE);
    T_LED_On(IN := FALSE);

    // Generate first random gap
    Rand_Gen(Execute := TRUE, Seed := 0, Rnd => RandN);
    IF RandN < 0.2 THEN
        T_Gap(PT := t#500ms);
    ELSIF RandN < 0.4 THEN
        T_Gap(PT := t#750ms);
    ELSIF RandN < 0.6 THEN
        T_Gap(PT := t#1000ms);
    ELSIF RandN < 0.8 THEN
        T_Gap(PT := t#1250ms);
    ELSE
        T_Gap(PT := t#1500ms);
    END_IF;
END_IF;

// Emergency stop
Trig_Mainreset(CLK := IBTN_MAIN AND GameActive AND NOT GameOver_Active);

IF Trig_Mainreset.Q THEN
    GameActive := FALSE;
    GameOver_Active := TRUE;
    GameOver_Step := 0;
    T_Seq(IN := FALSE, PT := t#300ms);
END_IF;

// Main game logic
IF GameActive THEN

    // Run 60 second timer
    T_GameTimer(IN := TRUE, PT := t#60s);

    // Time's up
    IF T_GameTimer.Q THEN
        GameActive := FALSE;
        GameOver_Active := TRUE;
        GameOver_Step := 0;
        T_Seq(IN := FALSE, PT := t#300ms);

        IF Score > HighScore THEN
            HighScore := Score;
        END_IF;
    END_IF;

    // GAP PHASE - waiting for LED (don't press anything!)
    IF GapActive THEN
        // All LEDs off
        OLED_Y := FALSE;
        OLED_B := FALSE;
        OLED_R := FALSE;
        CurrentLED := 0;

        // Run gap timer
        T_Gap(IN := TRUE);

        // Check for early button press
        Trig_Y(CLK := IBTN_Y);
        Trig_B(CLK := IBTN_B);
        Trig_R(CLK := IBTN_R);

        // Pressed during gap - instant game over
        IF Trig_Y.Q OR Trig_B.Q OR Trig_R.Q THEN
            GameActive := FALSE;
            GameOver_Active := TRUE;
            GameOver_Step := 0;
            T_Seq(IN := FALSE, PT := t#300ms);
            GapActive := FALSE;
            LEDActive := FALSE;
            T_Gap(IN := FALSE);
            T_LED_On(IN := FALSE);

            IF Score > HighScore THEN
                HighScore := Score;
            END_IF;
        END_IF;

        // Gap finished - light up random LED
        IF T_Gap.Q THEN
            T_Gap(IN := FALSE);
            GapActive := FALSE;
            LEDActive := TRUE;

            Rand_Gen(Execute := TRUE, Seed := 0, Rnd => RandN);
            CurrentLED := F_Rand(RandomValue := RandN);

            // Start 500ms timer
            T_LED_On(IN := FALSE, PT := t#500ms);
        END_IF;
    END_IF;

    // LED PHASE - press the correct button
    IF LEDActive THEN
        // Turn on the LED
        CASE CurrentLED OF
            1: OLED_Y := TRUE; OLED_B := FALSE; OLED_R := FALSE;
            2: OLED_Y := FALSE; OLED_B := TRUE; OLED_R := FALSE;
            3: OLED_Y := FALSE; OLED_B := FALSE; OLED_R := TRUE;
            ELSE OLED_Y := FALSE; OLED_B := FALSE; OLED_R := FALSE;
        END_CASE;

        // Run LED timer
        T_LED_On(IN := TRUE, PT := t#500ms);

        // Check button presses using the new function
        Trig_Y(CLK := IBTN_Y);
        Trig_B(CLK := IBTN_B);
        Trig_R(CLK := IBTN_R);

        // Handle all button presses with the function
        HandleButtonPress(
            ButtonPressed := Trig_Y.Q,
            ExpectedLED := 1,
            CurrentLED := CurrentLED,
            Score := Score,
            GameActive := GameActive,
            GameOver_Active := GameOver_Active,
            LEDActive := LEDActive,
            GapActive := GapActive,
            HighScore := HighScore,
            GameOver_Step := GameOver_Step,
            T_LED_On := T_LED_On,
            T_Gap := T_Gap,
            T_Seq := T_Seq,
            Rand_Gen := Rand_Gen,
            RandN := RandN
        );

        HandleButtonPress(
            ButtonPressed := Trig_B.Q,
            ExpectedLED := 2,
            CurrentLED := CurrentLED,
            Score := Score,
            GameActive := GameActive,
            GameOver_Active := GameOver_Active,
            LEDActive := LEDActive,
            GapActive := GapActive,
            HighScore := HighScore,
            GameOver_Step := GameOver_Step,
            T_LED_On := T_LED_On,
            T_Gap := T_Gap,
            T_Seq := T_Seq,
            Rand_Gen := Rand_Gen,
            RandN := RandN
        );

        HandleButtonPress(
            ButtonPressed := Trig_R.Q,
            ExpectedLED := 3,
            CurrentLED := CurrentLED,
            Score := Score,
            GameActive := GameActive,
            GameOver_Active := GameOver_Active,
            LEDActive := LEDActive,
            GapActive := GapActive,
            HighScore := HighScore,
            GameOver_Step := GameOver_Step,
            T_LED_On := T_LED_On,
            T_Gap := T_Gap,
            T_Seq := T_Seq,
            Rand_Gen := Rand_Gen,
            RandN := RandN
        );

        // Timer expired - too slow
        IF T_LED_On.Q THEN
            GameActive := FALSE;
            GameOver_Active := TRUE;
            GameOver_Step := 0;
            T_Seq(IN := FALSE, PT := t#300ms);
            LEDActive := FALSE;
            GapActive := FALSE;
            OLED_Y := FALSE;
            OLED_B := FALSE;
            OLED_R := FALSE;
            T_LED_On(IN := FALSE);
            T_Gap(IN := FALSE);

            IF Score > HighScore THEN
                HighScore := Score;
            END_IF;
        END_IF;
    END_IF;
END_IF;

// Game over animation using FB
IF GameOver_Active THEN
    GameOverA(
        Start := TRUE,
        Reset := FALSE
    );

    // Apply LED outputs
    OLED_Y := GameOverA.LED_Yellow;
    OLED_B := GameOverA.LED_Blue;
    OLED_R := GameOverA.LED_Red;

    // Check if animation done
    IF GameOverA.Done THEN
        GameOver_Active := FALSE;
        GameActive := FALSE;
        LEDActive := FALSE;
        GapActive := FALSE;
        Score := 0;
    END_IF;
ELSE
    // Reset animation when not in game over
    GameOverA(
        Start := FALSE,
        Reset := TRUE
    );
END_IF;

(* ---- simon_says_enhanced.st ---- *)
// Enhanced Simon Says with Sequence Display

// Variables for sequence display
VAR
    // Existing variables (keep all your existing ones)
    OLED_MAIN : BOOL;
    OLED_B : BOOL;
    OLED_R : BOOL;
    OLED_Y : BOOL;
    IBTN_MAIN : BOOL;
    IBTN_B : BOOL;
    IBTN_R : BOOL;
    IBTN_Y : BOOL;
    B : BOOL;
    RandN : REAL;
    L_N : INT;
    WriteIndex : INT := 0;
    ArrayFull : BOOL;
    Idx : INT;
    GameFlow_SN : ARRAY[0..49] OF INT;
    GameFlow_S : ARRAY[0..49] OF INT;
    ResetReq : BOOL;
    RI : BOOL;
    GameOver_Active : BOOL;
    GameOver_Step : INT;
    GameOver_Tick : BOOL;

    // New variables for sequence display
    SequenceDisplay_Active : BOOL := FALSE;
    SequenceDisplay_Index : INT := 0;
    SequenceDisplay_State : INT := 0; // 0=OFF, 1=ON
    CurrentRound : INT := 0;
    RoundStarted : BOOL := FALSE;

    // Timers
    T_Seq : TON;
    T_Display : TON;  // Timer for sequence display

    // Triggers
    Trig_Start : R_TRIG;
    Trig_Wrap : R_TRIG;
    Trig_Reset : R_TRIG;
    Trig_Tick : R_TRIG;
    Trig_DisplayTick : R_TRIG;
    Trig_RoundStart : R_TRIG;

    // Function blocks
    Rand_Gen : RAND;
    AryAddV : ARRAY_ADD;
END_VAR

// MAIN is N.C. → LED on when pressed
OLED_MAIN := NOT IBTN_MAIN;

// --- SEQUENCE DISPLAY LOGIC ---
// This runs before player input to show the sequence
IF SequenceDisplay_Active THEN
    // Timer for sequence display timing
    IF NOT T_Display.Q THEN
        IF SequenceDisplay_State = 0 THEN
            T_Display(IN := TRUE, PT := T#500ms);  // LED ON time
        ELSE
            T_Display(IN := TRUE, PT := T#300ms);  // LED OFF time between elements
        END_IF;
    ELSE
        T_Display(IN := FALSE);
    END_IF;

    Trig_DisplayTick(CLK := T_Display.Q);

    IF Trig_DisplayTick.Q THEN
        IF SequenceDisplay_State = 0 THEN
            // Turn ON the LED for current sequence element
            SequenceDisplay_State := 1;
        ELSE
            // Turn OFF and move to next element
            SequenceDisplay_State := 0;
            SequenceDisplay_Index := SequenceDisplay_Index + 1;

            // Check if we've displayed all elements for current round
            IF SequenceDisplay_Index >= CurrentRound THEN
                SequenceDisplay_Active := FALSE;
                SequenceDisplay_Index := 0;
                // Now player can start inputting
            END_IF;
        END_IF;
    END_IF;

    // Control LEDs based on sequence display
    IF SequenceDisplay_State = 1 AND SequenceDisplay_Index < CurrentRound THEN
        CASE GameFlow_SN[SequenceDisplay_Index] OF
            1: // Yellow
                OLED_Y := TRUE;
                OLED_B := FALSE;
                OLED_R := FALSE;
            2: // Blue
                OLED_Y := FALSE;
                OLED_B := TRUE;
                OLED_R := FALSE;
            3: // Red
                OLED_Y := FALSE;
                OLED_B := FALSE;
                OLED_R := TRUE;
            ELSE
                OLED_Y := FALSE;
                OLED_B := FALSE;
                OLED_R := FALSE;
        END_CASE;
    ELSE
        // Turn off all LEDs between sequence elements
        OLED_Y := FALSE;
        OLED_B := FALSE;
        OLED_R := FALSE;
    END_IF;

ELSIF NOT GameOver_Active THEN
    // Normal button → LED control (only when not displaying sequence or game over)
    OLED_B := IBTN_B;
    OLED_R := IBTN_R;
    OLED_Y := IBTN_Y;
END_IF;

// --- MAIN GAME LOGIC ---
Trig_Start(Clk := IBTN_B, Q => B);

IF B AND NOT SequenceDisplay_Active AND NOT GameOver_Active THEN
    // Generate random number for new sequence element
    Rand_Gen(Execute := TRUE, Seed := 0, Rnd => RandN);

    IF RandN < 0.333 THEN
        L_N := 1;  // Yellow
    ELSIF RandN < 0.666 THEN
        L_N := 2;  // Blue
    ELSE
        L_N := 3;  // Red
    END_IF;

    // Add to sequence array
    IF WriteIndex >= 50 THEN
        WriteIndex := 0;
        ArrayFull := TRUE;
    ELSIF WriteIndex < 0 THEN
        WriteIndex := 0;
    END_IF;

    Idx := TO_INT(WriteIndex);
    GameFlow_SN[Idx] := L_N;
    WriteIndex := WriteIndex + 1;

    // Update current round and trigger sequence display
    CurrentRound := WriteIndex;
    SequenceDisplay_Active := TRUE;
    SequenceDisplay_Index := 0;
    SequenceDisplay_State := 0;
    T_Display(IN := FALSE);  // Reset display timer
END_IF;

// --- RESET LOGIC ---
// Auto-reset edge when WriteIndex hits 50
Trig_Wrap(CLK := (WriteIndex = 50));
ResetReq := RI OR Trig_Wrap.Q;      // manual RI or auto edge at 50
Trig_Reset(CLK := ResetReq);

IF Trig_Reset.Q THEN
    AryAddV(In1 := GameFlow_S[0], In2 := L_N, Size := 50, AryOut := GameFlow_SN[0]);

    // Stop sequence display if active
    SequenceDisplay_Active := FALSE;
    SequenceDisplay_Index := 0;
    CurrentRound := 0;

    // Start game over sequence
    GameOver_Active := TRUE;
    GameOver_Step := -1;
    T_Seq(IN := FALSE, PT := T#300ms);

    WriteIndex := 0;
    ArrayFull := TRUE;
END_IF;

// --- GAME OVER LED SEQUENCE ---
IF GameOver_Active THEN
    IF NOT T_Seq.Q THEN
        T_Seq(IN := TRUE, PT := T#300ms);
    ELSE
        T_Seq(IN := FALSE, PT := T#300ms);
    END_IF;

    Trig_Tick(CLK := T_Seq.Q);
    GameOver_Tick := Trig_Tick.Q;

    IF GameOver_Tick THEN
        GameOver_Step := GameOver_Step + 1;
    END_IF;

    CASE GameOver_Step OF
        0:  OLED_R := TRUE;  OLED_B := FALSE; OLED_Y := FALSE;
        1:  OLED_R := FALSE; OLED_B := TRUE;  OLED_Y := FALSE;
        2:  OLED_R := FALSE; OLED_B := FALSE; OLED_Y := TRUE;
        4:  OLED_R := FALSE; OLED_B := FALSE; OLED_Y := FALSE;
        5:  OLED_R := TRUE;  OLED_B := TRUE;  OLED_Y := TRUE;
        6:  OLED_R := FALSE; OLED_B := FALSE; OLED_Y := FALSE;
        7:  OLED_R := TRUE;  OLED_B := TRUE;  OLED_Y := TRUE;
        ELSE
            OLED_R := FALSE; OLED_B := FALSE; OLED_Y := FALSE;
    END_CASE;

    IF GameOver_Step > 7 THEN
        GameOver_Active := FALSE;
        OLED_R := FALSE; OLED_B := FALSE; OLED_Y := FALSE;
    END_IF;
END_IF;
